FUNCTION_BLOCK FB_XY_PickAndPlace EXTENDS FB_ActionBasic
VAR_INPUT
	xExecute : BOOL;
	xAbort : BOOL;
	xReset :BOOL;
	AxisX_No : AxisNo;
	AxisY_No : AxisNo;
    TimeOut     : LREAL := 30; // Unit : s

END_VAR
VAR_OUTPUT
	xAborted : BOOL;
END_VAR
VAR
	StateBehavior :CBML.ETrigATo;
	Cylinder : REFERENCE TO UNI_CylinderList;
END_VAR

THIS^.IBehaviourModel := StateBehavior;
StateBehavior(
	xExecute:= xExecute, 
	xAbort:= xAbort, 
	udiTimeOut:= LREAL_TO_UDINT( TimeOut*1000000), 
	xDone=> xDone, 
	xBusy=> xBusy, 
	xError=> xError, 
	xAborted=> xAborted);

METHOD CleanupAction
VAR_INPUT
    xAbortProposed : BOOL;
    iErrorIDProposed: INT;
END_VAR
VAR_OUTPUT
    xComplete : BOOL := TRUE;
    xAbort: BOOL := xAbortProposed;
 	iErrorID : INT := iErrorIDProposed;
END_VAR
END_METHOD

METHOD CyclicAction
VAR_INPUT
    itfTimingController : CBML.ITimingController;
END_VAR
VAR_OUTPUT
    xComplete : BOOL := TRUE;
    iErrorID : INT := 0;
END_VAR
END_METHOD

METHOD ExitAction
VAR_INPUT
    xAfterCleanup : BOOL;
    xInCopyCode : BOOL;
END_VAR
END_METHOD

METHOD ResetAction
VAR_OUTPUT
    xComplete : BOOL := TRUE;
END_VAR
END_METHOD

METHOD StartAction
VAR_OUTPUT
    xComplete : BOOL := TRUE;
	iErrorID : INT := 0;
END_VAR
IF
END_METHOD

END_FUNCTION_BLOCK

(* stored: Version 1.1.0.1, ProductVersion 3.1.4024.13
   POU FB_XY_PickAndPlace: Id {1e0a96d6-7841-4417-a44d-529e52e8d9cb}, SpecialFunc None
   Folder Action: Id {a4922d67-fded-4fdb-9d35-1c066c0292b6}
   Method CleanupAction: Id {4e9acae2-331e-44ed-b279-f9a4e876f98e}
   Method CyclicAction: Id {0d7405f8-15ab-40ec-895a-632aaf42a80f}
   Method ExitAction: Id {5648775b-4d62-4adf-b354-517acc9cb63d}
   Method ResetAction: Id {341a82f5-f15b-423a-92c4-10f7b0afb693}
   Method StartAction: Id {a9ee3687-40a3-44e9-8da7-161b241adaf9} *)
